// TIA Portal V19 export
VAR_GLOBAL   // PLC tag table "Global"
END_VAR
